PROGRAM INPUTS (*: INT*)
VAR

	EN1000_IO_StatusTON :TON;
	//NRHMIS_IO_StatusTON :TON;
	//NRHMI_Heartbeat_TON: TON;
	//NRHMI_INT: INT:=0;
	//NRHMI_Heartbeat_Last: BOOL:=0;

	SYSDATA_Heartbeat_TON: TON;
	SYSDATA_INT: INT:=0;
	SYSDATA_Heartbeat_Last: BOOL:=0;
	
	SYSDATA_Heartbeat_TON2: TON;
	SYSDATA_INT2: INT:=0;
	SYSDATA_Heartbeat_Last2: BOOL:=0;

	//DV1501_Manip_Rot_ErrorTON :TON;

	TEMP:UDINT:=0;
	temp1:REAL:=0;
	temp2:REAL:=0;
	
	PI : REAL := 3.14159;
	
END_VAR
VAR_INPUT

(*
//NEAR REMOTE HMI STATION I/O	
	//Communication Status
		RIO2022_Status AT %I*: BOOL;
	//Digital Input Module
		RIO1919_DI1 AT %I*: BOOL; RIO1919_DI2 AT %I*: BOOL; RIO1919_DI3 AT %I*: BOOL; RIO1919_DI4 AT %I*: BOOL; RIO1919_DI5 AT %I*: BOOL; RIO1919_DI6 AT %I*: BOOL; RIO1919_DI7 AT %I*: BOOL; RIO1919_DI8 AT %I*: BOOL;
	//Analog Input Module
		RIO1924_AI1 AT %I*: INT; RIO1924_AI2 AT %I*: INT; RIO1924_AI3 AT %I*: INT; RIO1924_AI4 AT %I*: INT;
		RIO1926_AI1 AT %I*: INT; RIO1926_AI2 AT %I*: INT; RIO1926_AI3 AT %I*: INT; RIO1926_AI4 AT %I*: INT;
		RIO1928A_AI1 AT %I*: INT; RIO1928A_AI2 AT %I*: INT; RIO1928A_AI3 AT %I*: INT; RIO1928A_AI4 AT %I*: INT;
	//Subscribe VAR
		NRHMI_SYS_SUB1 AT %I*: MAIN_P_7;
*)

//EN1000 
	//Communication Status
		//RIO1102_Status AT %I*: BOOL;
	//Digital Input Module
		RIO1108_DI1 AT %I*: BOOL; RIO1108_DI2 AT %I*: BOOL; RIO1108_DI3 AT %I*: BOOL; RIO1108_DI4 AT %I*: BOOL; RIO1108_DI5 AT %I*: BOOL; RIO1108_DI6 AT %I*: BOOL; RIO1108_DI7 AT %I*: BOOL; RIO1108_DI8 AT %I*: BOOL;
		RIO1110_DI1 AT %I*: BOOL; RIO1110_DI2 AT %I*: BOOL; RIO1110_DI3 AT %I*: BOOL; RIO1110_DI4 AT %I*: BOOL; RIO1110_DI5 AT %I*: BOOL; RIO1110_DI6 AT %I*: BOOL; RIO1110_DI7 AT %I*: BOOL; RIO1110_DI8 AT %I*: BOOL;
		RIO1112_DI1 AT %I*: BOOL; RIO1112_DI2 AT %I*: BOOL; RIO1112_DI3 AT %I*: BOOL; RIO1112_DI4 AT %I*: BOOL; RIO1112_DI5 AT %I*: BOOL; RIO1112_DI6 AT %I*: BOOL; RIO1112_DI7 AT %I*: BOOL; RIO1112_DI8 AT %I*: BOOL;
		RIO1114_DI1 AT %I*: BOOL; RIO1114_DI2 AT %I*: BOOL; RIO1114_DI3 AT %I*: BOOL; RIO1114_DI4 AT %I*: BOOL; RIO1114_DI5 AT %I*: BOOL;
	//Analog Input Module
		RIO1116_AI1 AT %I*: INT; RIO1116_AI2 AT %I*: INT; 
	
	// Resitor Bridge Module
		RIO1125_AI1 AT %I*: INT;
		RIO1127_AI1 AT %I*: INT;
		RIO1129_AI1 AT %I*: INT;
	
	//Servo Module (Resolver Input)
		RIO1137_AI1 AT %I*: UDINT;
		
	//Stepper Motor Modules
		RIO1135_ERROR AT %I*: BOOL;
		
	//Subscribe VAR
		//NRHMI_SUB AT %I*: NR_HMI_P_1;

END_VAR
VAR_OUTPUT
	
END_VAR

VAR_IN_OUT
	RGP: System;
	TS_IN: Touchscreen;
END_VAR

IF (INPUTS.RGP.PROG.LAPTOP_TEST_ENABLE=0) THEN
//NEAR REMOTE HMI STATION INPUTS
	(*	IF (RGP.PROG.Program_Location = 1) THEN 
			RGP.EN1900_NRHMI.PB1905_EMER_STOP:=RIO1919_DI1;
			RGP.EN1900_NRHMI.SS1940_DISABLE_NRCONTROL:=RIO1919_DI3;
			RGP.EN1900_NRHMI.SS1940_REQUEST_NRCONTROL:=RIO1919_DI4;
			
			NRHMIS_IO_StatusTON.PT:=T#0MS;
			IF ( NOT RIO2022_Status) THEN
				NRHMIS_IO_StatusTON.IN:=1;
			ELSE
				NRHMIS_IO_StatusTON.IN:=0;
			END_IF
			RGP.EN1900_NRHMI.EN1900_HEALTHY := NRHMIS_IO_StatusTON.Q;
			//NRHMIS_IO_StatusTON();
	
			RGP.EN1900_NRHMI.DV1917_JS_X_AXIS.SIGNAL.Raw_Data := INT_TO_REAL(RIO1928A_AI2);
			Joystick(JS:=RGP.EN1900_NRHMI.DV1917_JS_X_AXIS);
			RGP.EN1900_NRHMI.DV1917_JS_Y_AXIS.SIGNAL.Raw_Data := -INT_TO_REAL(RIO1928A_AI1);
			Joystick(JS:=RGP.EN1900_NRHMI.DV1917_JS_Y_AXIS);
			RGP.EN1900_NRHMI.DV1917_JS_Z_AXIS.SIGNAL.Raw_Data := INT_TO_REAL(RIO1924_AI4);
			Joystick(JS:=RGP.EN1900_NRHMI.DV1917_JS_Z_AXIS);
			
			RGP.EN1900_NRHMI.DV1927_JS_X_AXIS.SIGNAL.Raw_Data := INT_TO_REAL(RIO1924_AI2);
			Joystick(JS:=RGP.EN1900_NRHMI.DV1927_JS_X_AXIS);
			RGP.EN1900_NRHMI.DV1927_JS_Y_AXIS.SIGNAL.Raw_Data := -INT_TO_REAL(RIO1924_AI1);
			Joystick(JS:=RGP.EN1900_NRHMI.DV1927_JS_Y_AXIS);
			RGP.EN1900_NRHMI.DV1927_JS_Z_AXIS.SIGNAL.Raw_Data := INT_TO_REAL(RIO1924_AI3);
			Joystick(JS:=RGP.EN1900_NRHMI.DV1927_JS_Z_AXIS);
			
			RGP.EN1900_NRHMI.DV1938_JS_X_AXIS.SIGNAL.Raw_Data := INT_TO_REAL(RIO1926_AI2);
			Joystick(JS:=RGP.EN1900_NRHMI.DV1938_JS_X_AXIS);
			RGP.EN1900_NRHMI.DV1938_JS_Y_AXIS.SIGNAL.Raw_Data := -INT_TO_REAL(RIO1926_AI1);
			Joystick(JS:=RGP.EN1900_NRHMI.DV1938_JS_Y_AXIS);
			RGP.EN1900_NRHMI.DV1938_JS_Z_AXIS.SIGNAL.Raw_Data := INT_TO_REAL(RIO1926_AI3);
			Joystick(JS:=RGP.EN1900_NRHMI.DV1938_JS_Z_AXIS);
	
			//SYSTEM Data Monitor
				SYSDATA_Heartbeat_TON.PT := T#400MS;
				IF (SYSDATA_Heartbeat_Last <> NRHMI_SYS_SUB1.Heartbeat) THEN
					SYSDATA_Heartbeat_TON.IN:=0;
					IF (SYSDATA_INT < 10) THEN
						SYSDATA_INT := SYSDATA_INT+1;				
					ELSE
						RGP.PROG.HMI_FRMDATA_Heartbeat_Healthy:=1;
					END_IF
					SYSDATA_Heartbeat_Last := NRHMI_SYS_SUB1.Heartbeat;
				ELSE
					SYSDATA_Heartbeat_TON.IN:=1;
				END_IF
				IF (SYSDATA_Heartbeat_TON.Q) THEN
					RGP.PROG.HMI_FRMDATA_Heartbeat_Healthy:=0;
					SYSDATA_INT := 0;				
				END_IF
				SYSDATA_Heartbeat_TON();
	
				SYSDATA_Heartbeat_TON2.PT := T#400MS;
				//IF (SYSDATA_Heartbeat_Last2 <> NRHMI_SYS_SUB2.Heartbeat) THEN
				//	SYSDATA_Heartbeat_TON2.IN:=0;
				//	IF (SYSDATA_INT2 < 10) THEN
				//		SYSDATA_INT2 := SYSDATA_INT2+1;				
				//	ELSE
				//		RGP.PROG.HMI_FRMDATA2_Heartbeat_Healthy:=1;
				//	END_IF
				//	SYSDATA_Heartbeat_Last2 := NRHMI_SYS_SUB2.Heartbeat;
				//ELSE
				//	SYSDATA_Heartbeat_TON2.IN:=1;
				//END_IF
				//IF (SYSDATA_Heartbeat_TON2.Q) THEN
				//	RGP.PROG.HMI_FRMDATA2_Heartbeat_Healthy:=0;
				//END_IF
				//SYSDATA_Heartbeat_TON2();
	
			MAIN_SUB_TO_STR(RGP,NRHMI_SYS_SUB1, TS_IN);
	*)
// ELSIF (RGP.PROG.Program_Location = 0) THEN //EN1000		// Uncomment if using Remote HMI
	
	IF (RGP.PROG.Program_Location = 0) THEN //EN1000

		// E-Stop & Safety
			RGP.EN1000.DV1052_SMR:=RIO1114_DI5;
		
		// Selector Switches		
			RGP.EN1000.SS1338_POS_TOOL_ROTZ_POS := RIO1112_DI1;
			RGP.EN1000.SS1338_POS_TOOL_ROTZ_NEG := RIO1112_DI2;
			RGP.EN1000.SS1157_TRANSX_POS := RIO1108_DI1;
			RGP.EN1000.SS1157_TRANSX_NEG := RIO1108_DI2;
			RGP.EN1000.SS1182_TRANSY_POS := RIO1108_DI3;
			RGP.EN1000.SS1182_TRANSY_NEG := RIO1108_DI4;
			RGP.EN1000.SS1264_ALL_JACKS_TRANSZ_POS := RIO1108_DI5;
			RGP.EN1000.SS1264_ALL_JACKS_TRANSZ_NEG := RIO1108_DI6;
			RGP.EN1000.SS1307_JACK1_TRANSZ_POS := RIO1110_DI3;
			RGP.EN1000.SS1307_JACK1_TRANSZ_NEG := RIO1110_DI4;
			RGP.EN1000.SS1312_JACK2_TRANSZ_POS := RIO1110_DI5;
			RGP.EN1000.SS1312_JACK2_TRANSZ_NEG := RIO1110_DI6;
			RGP.EN1000.SS1324_JACK3_TRANSZ_POS := RIO1110_DI7;
			RGP.EN1000.SS1324_JACK3_TRANSZ_NEG := RIO1110_DI8;
			RGP.EN1000.SS1273_TILT_ROTX_POS := RIO1108_DI7;
			RGP.EN1000.SS1273_TILT_ROTX_NEG := RIO1108_DI8;
			RGP.EN1000.SS1282_TILT_ROTY_POS := RIO1110_DI1;
			RGP.EN1000.SS1282_TILT_ROTY_NEG := RIO1110_DI2;
			RGP.EN1000.SS1457_MON_TOOL_ROTZ_POS := RIO1114_DI3;
			RGP.EN1000.SS1457_MON_TOOL_ROTZ_NEG := RIO1114_DI4;
				
		// Limit Switches (EOT)
			RGP.EN1000.LS1352_JACK1_EOT_POS := NOT RIO1112_DI3;
			RGP.EN1000.DV1151_JACK1_DRIVE.IN_EOT_POS := RGP.EN1000.LS1352_JACK1_EOT_POS;
			RGP.EN1000.LS1354_JACK1_EOT_NEG := NOT RIO1112_DI4;
			RGP.EN1000.DV1151_JACK1_DRIVE.IN_EOT_NEG := RGP.EN1000.LS1354_JACK1_EOT_NEG; 
			
			RGP.EN1000.LS1357_JACK2_EOT_POS := NOT RIO1112_DI5;
			RGP.EN1000.DV1275_JACK2_DRIVE.IN_EOT_POS := RGP.EN1000.LS1357_JACK2_EOT_POS;
			RGP.EN1000.LS1359_JACK2_EOT_NEG := NOT RIO1112_DI6;
			RGP.EN1000.DV1275_JACK2_DRIVE.IN_EOT_NEG := RGP.EN1000.LS1359_JACK2_EOT_NEG;
	 
			RGP.EN1000.LS1362_JACK3_EOT_POS := NOT RIO1112_DI7;
			RGP.EN1000.DV1301_JACK3_DRIVE.IN_EOT_POS := RGP.EN1000.LS1362_JACK3_EOT_POS;
			RGP.EN1000.LS1364_JACK3_EOT_NEG := NOT RIO1112_DI8;
			RGP.EN1000.DV1301_JACK3_DRIVE.IN_EOT_NEG := RGP.EN1000.LS1364_JACK3_EOT_NEG;
			
			RGP.EN1000.LS1367_POS_TOOL_ROTZ_EOT_POS := NOT RIO1114_DI1; // 0 SIGNAL MEANS EOT HAS BEEN TRIPPED
			RGP.EN1000.DV1325_POS_TOOL_ROTZ_DRIVE.IN_EOT_POS := RGP.EN1000.LS1367_POS_TOOL_ROTZ_EOT_POS;
			RGP.EN1000.LS1369_POS_TOOL_ROTZ_EOT_NEG := NOT RIO1114_DI2;
			RGP.EN1000.DV1325_POS_TOOL_ROTZ_DRIVE.IN_EOT_NEG := RGP.EN1000.LS1369_POS_TOOL_ROTZ_EOT_NEG;				
			
		// Tilt Sensors	
			RGP.EN1000.DV1390_TILT_SENSOR1.Raw_Data := INT_TO_REAL(RIO1116_AI1);  
			Analog_In(AI:=RGP.EN1000.DV1390_TILT_SENSOR1);
			
			RGP.EN1000.DV1396_TILT_SENSOR2.Raw_Data := INT_TO_REAL(RIO1116_AI2);  
			Analog_In(AI:=RGP.EN1000.DV1396_TILT_SENSOR2);
			
		// Load Cells
			RGP.EN1000.DV1375_LOAD_CELL_JACK1_FZ.Raw_Data := INT_TO_REAL(RIO1125_AI1);
			Analog_In(AI:=RGP.EN1000.DV1375_LOAD_CELL_JACK1_FZ);
			
			RGP.EN1000.DV1379_LOAD_CELL_JACK2_FZ.Raw_Data := INT_TO_REAL(RIO1127_AI1);
			Analog_In(AI:=RGP.EN1000.DV1379_LOAD_CELL_JACK2_FZ);
			
			RGP.EN1000.DV1385_LOAD_CELL_JACK3_FZ.Raw_Data := INT_TO_REAL(RIO1129_AI1);
			Analog_In(AI:=RGP.EN1000.DV1385_LOAD_CELL_JACK3_FZ);
		
		// Resolvers
			// X-TRANS			//FIXME: NEEDED FOR DISPLAY??
				//TEMP:= ??? ; TEMP.20:=0; TEMP.21:=0; TEMP.22:=0; TEMP.23:=0; TEMP.24:=0; TEMP.25:=0; TEMP.26:=0; TEMP.27:=0; TEMP.28:=0; TEMP.29:=0; TEMP.30:=0; TEMP.31:=0;
				//RGP.EN1000.DV1150_TRANSX_DRIVE.Feedback.Raw_Data := UDINT_TO_REAL(TEMP);
				//Axis_Pos(RGP.EN1000.DV1150_TRANSX_DRIVE.Feedback,RGP.PROG.delT,RGP.PROG.calculate);
			
			// Y-TRANS			//FIXME: NEEDED FOR DISPLAY??
				//TEMP:= ??? ; TEMP.20:=0; TEMP.21:=0; TEMP.22:=0; TEMP.23:=0; TEMP.24:=0; TEMP.25:=0; TEMP.26:=0; TEMP.27:=0; TEMP.28:=0; TEMP.29:=0; TEMP.30:=0; TEMP.31:=0;
				//RGP.EN1000.DV1175_TRANSY_DRIVE.Feedback.Raw_Data := UDINT_TO_REAL(TEMP);
				//Axis_Pos(RGP.EN1000.DV1175_TRANSY_DRIVE.Feedback,RGP.PROG.delT,RGP.PROG.calculate);
				
			// JACK 1
				//TEMP:= ??? ; TEMP.20:=0; TEMP.21:=0; TEMP.22:=0; TEMP.23:=0; TEMP.24:=0; TEMP.25:=0; TEMP.26:=0; TEMP.27:=0; TEMP.28:=0; TEMP.29:=0; TEMP.30:=0; TEMP.31:=0;
				//RGP.EN1000.DV1151_JACK1_DRIVE.Feedback.Raw_Data := UDINT_TO_REAL(TEMP);
				Axis_Pos(RGP.EN1000.DV1151_JACK1_DRIVE.Feedback,RGP.PROG.delT,RGP.PROG.calculate);
			
			// JACK 2
				//TEMP:= ??? ; TEMP.20:=0; TEMP.21:=0; TEMP.22:=0; TEMP.23:=0; TEMP.24:=0; TEMP.25:=0; TEMP.26:=0; TEMP.27:=0; TEMP.28:=0; TEMP.29:=0; TEMP.30:=0; TEMP.31:=0;
				//RGP.EN1000.DV1275_JACK2_DRIVE.Feedback.Raw_Data := UDINT_TO_REAL(TEMP);
				Axis_Pos(RGP.EN1000.DV1275_JACK2_DRIVE.Feedback,RGP.PROG.delT,RGP.PROG.calculate);
			
			// JACK 3
				//TEMP:= ??? ; TEMP.20:=0; TEMP.21:=0; TEMP.22:=0; TEMP.23:=0; TEMP.24:=0; TEMP.25:=0; TEMP.26:=0; TEMP.27:=0; TEMP.28:=0; TEMP.29:=0; TEMP.30:=0; TEMP.31:=0;
				//RGP.EN1000.DV1301_JACK3_DRIVE.Feedback.Raw_Data := UDINT_TO_REAL(TEMP);
				Axis_Pos(RGP.EN1000.DV1301_JACK3_DRIVE.Feedback,RGP.PROG.delT,RGP.PROG.calculate);
			
			// POS TOOL ROT-Z
				//TEMP:= ??? ; TEMP.20:=0; TEMP.21:=0; TEMP.22:=0; TEMP.23:=0; TEMP.24:=0; TEMP.25:=0; TEMP.26:=0; TEMP.27:=0; TEMP.28:=0; TEMP.29:=0; TEMP.30:=0; TEMP.31:=0;
				//RGP.EN1000.DV1325_POS_TOOL_ROTZ_DRIVE.Feedback.Raw_Data := UDINT_TO_REAL(TEMP); 
				Axis_Pos(RGP.EN1000.DV1325_POS_TOOL_ROTZ_DRIVE.Feedback,RGP.PROG.delT,RGP.PROG.calculate);
			
			// MON TOOL ROT-Z
				TEMP:=RIO1137_AI1; TEMP.20:=0; TEMP.21:=0; TEMP.22:=0; TEMP.23:=0; TEMP.24:=0; TEMP.25:=0; TEMP.26:=0; TEMP.27:=0; TEMP.28:=0; TEMP.29:=0; TEMP.30:=0; TEMP.31:=0;
				RGP.EN1000.RIO1135_MON_TOOL_ROTZ_DRIVE.Feedback.Raw_Data := UDINT_TO_REAL(TEMP);  
				Axis_Pos(RGP.EN1000.RIO1135_MON_TOOL_ROTZ_DRIVE.Feedback,RGP.PROG.delT,RGP.PROG.calculate);
						
		// Tilt Control
			// Jack's Angle about Z
		 		RGP.PROG.JACK1_ANGLE_ABOUT_Z := 0;					// FIXME: CONVERT RESOLVER COUNTS TO DEGREE VALUE
				RGP.PROG.JACK2_ANGLE_ABOUT_Z := RGP.PROG.JACK1_ANGLE_ABOUT_Z + 120;
				RGP.PROG.JACK3_ANGLE_ABOUT_Z := RGP.PROG.JACK1_ANGLE_ABOUT_Z + 240;
							
			// X-Position  
				RGP.PROG.JACK1_X_POSITION := RGP.PROG.POS_TOOL_RADIUS*COS(RGP.PROG.JACK1_ANGLE_ABOUT_Z/(180*PI));
				RGP.PROG.JACK2_X_POSITION := RGP.PROG.POS_TOOL_RADIUS*COS(RGP.PROG.JACK2_ANGLE_ABOUT_Z/(180*PI));
				RGP.PROG.JACK3_X_POSITION := RGP.PROG.POS_TOOL_RADIUS*COS(RGP.PROG.JACK3_ANGLE_ABOUT_Z/(180*PI));
			
			// Y-Position 
				RGP.PROG.JACK1_Y_POSITION := RGP.PROG.POS_TOOL_RADIUS*SIN(RGP.PROG.JACK1_ANGLE_ABOUT_Z/(180*PI));
				RGP.PROG.JACK2_Y_POSITION := RGP.PROG.POS_TOOL_RADIUS*SIN(RGP.PROG.JACK2_ANGLE_ABOUT_Z/(180*PI));
				RGP.PROG.JACK3_Y_POSITION := RGP.PROG.POS_TOOL_RADIUS*SIN(RGP.PROG.JACK3_ANGLE_ABOUT_Z/(180*PI));
				
			// Z-Position 
				RGP.PROG.JACK1_Z_POSITION := RGP.EN1000.DV1151_JACK1_DRIVE.Feedback.Position;
				RGP.PROG.JACK2_Z_POSITION := RGP.EN1000.DV1275_JACK2_DRIVE.Feedback.Position;
				RGP.PROG.JACK3_Z_POSITION := RGP.EN1000.DV1301_JACK3_DRIVE.Feedback.Position;		

	END_IF
END_IF

END_PROGRAM

(* stored: Version 1.1.0.1, ProductVersion 3.1.4024.0
   POU INPUTS: Id {ec4607e6-a585-45f3-bd52-6ea7ddee2e87}, SpecialFunc None *)
